// TIA Portal V17 export
// export: Created 2025-03-12T15:33:26.3402527Z, ExportSetting WithDefaults, DisplayName Totally Integrated Automation Portal, DisplayVersion V17 Update 8, DisplayName TIA Portal Openness, DisplayVersion V17 Update 8, DisplayName TIA Portal Version Control Interface, DisplayVersion V17, DisplayName SINAMICS Startdrive Advanced, DisplayVersion V17 SP2, DisplayName SINAMICS Startdrive G110M, G120, G120C, G120D, G120P, G115D, DisplayVersion V17 SP2, DisplayName SINAMICS Startdrive G130, G150, S120, S150, SINAMICS MV, S210, DisplayVersion V17 SP2, DisplayName STEP 7 Professional, DisplayVersion V17 Update 8, DisplayName SINUMERIK ONE STEP 7 Toolbox, DisplayVersion V17 Update 12, DisplayName SINUMERIK 840D sl STEP 7 Toolbox, DisplayVersion V17 Update 12, DisplayName STEP 7 Safety, DisplayVersion V17 Update 6, DisplayName WinCC Advanced, DisplayVersion V17 Update 8
FUNCTION "FC7339_ROBOT_CELL_TEST_INTERLOCK" : Void   // FC7339, LAD
{ S7_Optimized_Access := 'FALSE' }
AUTHOR : ETXETAR
VERSION : 1.0
// stored: AutoNumber false, IsIECCheckEnabled false, SetENOAutomatically false, UDAEnableTagReadback false
   VAR_TEMP
      RETVAL_1 : Int;
   END_VAR
BEGIN

REGION Network 1: ROBOT HEARTBEAT / STOP AT END OF CYCLE
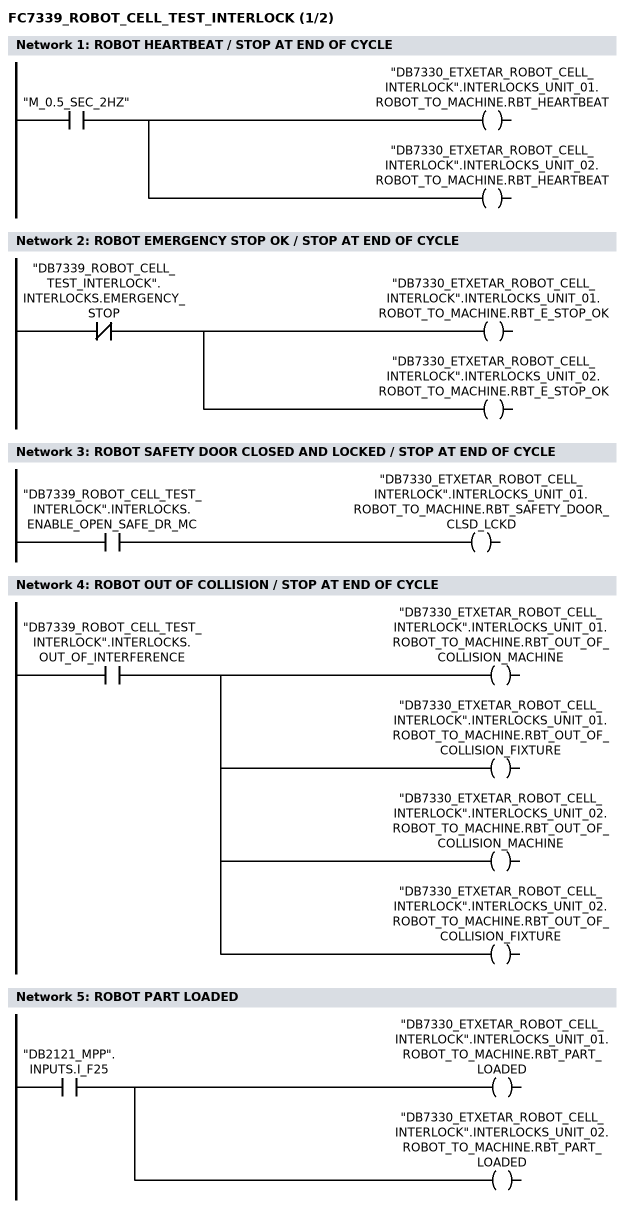
   RUNG wire#powerrail
      Contact( "M_0.5_SEC_2HZ" )
      wire#w1
      Coil( "DB7330_ETXETAR_ROBOT_CELL_INTERLOCK".INTERLOCKS_UNIT_01.ROBOT_TO_MACHINE.RBT_HEARTBEAT )
   END_RUNG
   RUNG wire#w1
      Coil( "DB7330_ETXETAR_ROBOT_CELL_INTERLOCK".INTERLOCKS_UNIT_02.ROBOT_TO_MACHINE.RBT_HEARTBEAT )
   END_RUNG
   // the same network as SCL:
   "DB7330_ETXETAR_ROBOT_CELL_INTERLOCK".INTERLOCKS_UNIT_01.ROBOT_TO_MACHINE.RBT_HEARTBEAT := "M_0.5_SEC_2HZ";
   "DB7330_ETXETAR_ROBOT_CELL_INTERLOCK".INTERLOCKS_UNIT_02.ROBOT_TO_MACHINE.RBT_HEARTBEAT := "M_0.5_SEC_2HZ";
END_REGION

REGION Network 2: ROBOT EMERGENCY STOP OK / STOP AT END OF CYCLE
   RUNG wire#powerrail
      I_Contact( "DB7339_ROBOT_CELL_TEST_INTERLOCK".INTERLOCKS.EMERGENCY_STOP )
      wire#w1
      Coil( "DB7330_ETXETAR_ROBOT_CELL_INTERLOCK".INTERLOCKS_UNIT_01.ROBOT_TO_MACHINE.RBT_E_STOP_OK )
   END_RUNG
   RUNG wire#w1
      Coil( "DB7330_ETXETAR_ROBOT_CELL_INTERLOCK".INTERLOCKS_UNIT_02.ROBOT_TO_MACHINE.RBT_E_STOP_OK )
   END_RUNG
   // the same network as SCL:
   "DB7330_ETXETAR_ROBOT_CELL_INTERLOCK".INTERLOCKS_UNIT_01.ROBOT_TO_MACHINE.RBT_E_STOP_OK := NOT "DB7339_ROBOT_CELL_TEST_INTERLOCK".INTERLOCKS.EMERGENCY_STOP;
   "DB7330_ETXETAR_ROBOT_CELL_INTERLOCK".INTERLOCKS_UNIT_02.ROBOT_TO_MACHINE.RBT_E_STOP_OK := NOT "DB7339_ROBOT_CELL_TEST_INTERLOCK".INTERLOCKS.EMERGENCY_STOP;
END_REGION

REGION Network 3: ROBOT SAFETY DOOR CLOSED AND LOCKED / STOP AT END OF CYCLE
   RUNG wire#powerrail
      Contact( "DB7339_ROBOT_CELL_TEST_INTERLOCK".INTERLOCKS.ENABLE_OPEN_SAFE_DR_MC )
      Coil( "DB7330_ETXETAR_ROBOT_CELL_INTERLOCK".INTERLOCKS_UNIT_01.ROBOT_TO_MACHINE.RBT_SAFETY_DOOR_CLSD_LCKD )
   END_RUNG
   // the same network as SCL:
   "DB7330_ETXETAR_ROBOT_CELL_INTERLOCK".INTERLOCKS_UNIT_01.ROBOT_TO_MACHINE.RBT_SAFETY_DOOR_CLSD_LCKD := "DB7339_ROBOT_CELL_TEST_INTERLOCK".INTERLOCKS.ENABLE_OPEN_SAFE_DR_MC;
END_REGION

REGION Network 4: ROBOT OUT OF COLLISION / STOP AT END OF CYCLE
   RUNG wire#powerrail
      Contact( "DB7339_ROBOT_CELL_TEST_INTERLOCK".INTERLOCKS.OUT_OF_INTERFERENCE )
      wire#w1
      Coil( "DB7330_ETXETAR_ROBOT_CELL_INTERLOCK".INTERLOCKS_UNIT_01.ROBOT_TO_MACHINE.RBT_OUT_OF_COLLISION_MACHINE )
   END_RUNG
   RUNG wire#w1
      Coil( "DB7330_ETXETAR_ROBOT_CELL_INTERLOCK".INTERLOCKS_UNIT_01.ROBOT_TO_MACHINE.RBT_OUT_OF_COLLISION_FIXTURE )
   END_RUNG
   RUNG wire#w1
      Coil( "DB7330_ETXETAR_ROBOT_CELL_INTERLOCK".INTERLOCKS_UNIT_02.ROBOT_TO_MACHINE.RBT_OUT_OF_COLLISION_MACHINE )
   END_RUNG
   RUNG wire#w1
      Coil( "DB7330_ETXETAR_ROBOT_CELL_INTERLOCK".INTERLOCKS_UNIT_02.ROBOT_TO_MACHINE.RBT_OUT_OF_COLLISION_FIXTURE )
   END_RUNG
   // the same network as SCL:
   "DB7330_ETXETAR_ROBOT_CELL_INTERLOCK".INTERLOCKS_UNIT_01.ROBOT_TO_MACHINE.RBT_OUT_OF_COLLISION_MACHINE := "DB7339_ROBOT_CELL_TEST_INTERLOCK".INTERLOCKS.OUT_OF_INTERFERENCE;
   "DB7330_ETXETAR_ROBOT_CELL_INTERLOCK".INTERLOCKS_UNIT_01.ROBOT_TO_MACHINE.RBT_OUT_OF_COLLISION_FIXTURE := "DB7339_ROBOT_CELL_TEST_INTERLOCK".INTERLOCKS.OUT_OF_INTERFERENCE;
   "DB7330_ETXETAR_ROBOT_CELL_INTERLOCK".INTERLOCKS_UNIT_02.ROBOT_TO_MACHINE.RBT_OUT_OF_COLLISION_MACHINE := "DB7339_ROBOT_CELL_TEST_INTERLOCK".INTERLOCKS.OUT_OF_INTERFERENCE;
   "DB7330_ETXETAR_ROBOT_CELL_INTERLOCK".INTERLOCKS_UNIT_02.ROBOT_TO_MACHINE.RBT_OUT_OF_COLLISION_FIXTURE := "DB7339_ROBOT_CELL_TEST_INTERLOCK".INTERLOCKS.OUT_OF_INTERFERENCE;
END_REGION

REGION Network 5: ROBOT PART LOADED
   RUNG wire#powerrail
      Contact( "DB2121_MPP".INPUTS.I_F25 )
      wire#w1
      Coil( "DB7330_ETXETAR_ROBOT_CELL_INTERLOCK".INTERLOCKS_UNIT_01.ROBOT_TO_MACHINE.RBT_PART_LOADED )
   END_RUNG
   RUNG wire#w1
      Coil( "DB7330_ETXETAR_ROBOT_CELL_INTERLOCK".INTERLOCKS_UNIT_02.ROBOT_TO_MACHINE.RBT_PART_LOADED )
   END_RUNG
   // the same network as SCL:
   "DB7330_ETXETAR_ROBOT_CELL_INTERLOCK".INTERLOCKS_UNIT_01.ROBOT_TO_MACHINE.RBT_PART_LOADED := "DB2121_MPP".INPUTS.I_F25;
   "DB7330_ETXETAR_ROBOT_CELL_INTERLOCK".INTERLOCKS_UNIT_02.ROBOT_TO_MACHINE.RBT_PART_LOADED := "DB2121_MPP".INPUTS.I_F25;
END_REGION

REGION Network 6: ROBOT PART UNLOADED
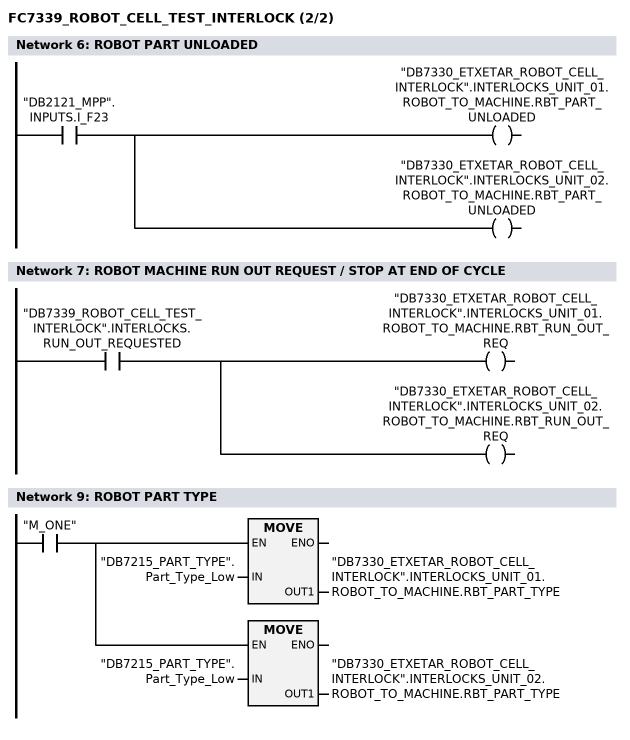
   RUNG wire#powerrail
      Contact( "DB2121_MPP".INPUTS.I_F23 )
      wire#w1
      Coil( "DB7330_ETXETAR_ROBOT_CELL_INTERLOCK".INTERLOCKS_UNIT_01.ROBOT_TO_MACHINE.RBT_PART_UNLOADED )
   END_RUNG
   RUNG wire#w1
      Coil( "DB7330_ETXETAR_ROBOT_CELL_INTERLOCK".INTERLOCKS_UNIT_02.ROBOT_TO_MACHINE.RBT_PART_UNLOADED )
   END_RUNG
   // the same network as SCL:
   "DB7330_ETXETAR_ROBOT_CELL_INTERLOCK".INTERLOCKS_UNIT_01.ROBOT_TO_MACHINE.RBT_PART_UNLOADED := "DB2121_MPP".INPUTS.I_F23;
   "DB7330_ETXETAR_ROBOT_CELL_INTERLOCK".INTERLOCKS_UNIT_02.ROBOT_TO_MACHINE.RBT_PART_UNLOADED := "DB2121_MPP".INPUTS.I_F23;
END_REGION

REGION Network 7: ROBOT MACHINE RUN OUT REQUEST / STOP AT END OF CYCLE
   RUNG wire#powerrail
      Contact( "DB7339_ROBOT_CELL_TEST_INTERLOCK".INTERLOCKS.RUN_OUT_REQUESTED )
      wire#w1
      Coil( "DB7330_ETXETAR_ROBOT_CELL_INTERLOCK".INTERLOCKS_UNIT_01.ROBOT_TO_MACHINE.RBT_RUN_OUT_REQ )
   END_RUNG
   RUNG wire#w1
      Coil( "DB7330_ETXETAR_ROBOT_CELL_INTERLOCK".INTERLOCKS_UNIT_02.ROBOT_TO_MACHINE.RBT_RUN_OUT_REQ )
   END_RUNG
   // the same network as SCL:
   "DB7330_ETXETAR_ROBOT_CELL_INTERLOCK".INTERLOCKS_UNIT_01.ROBOT_TO_MACHINE.RBT_RUN_OUT_REQ := "DB7339_ROBOT_CELL_TEST_INTERLOCK".INTERLOCKS.RUN_OUT_REQUESTED;
   "DB7330_ETXETAR_ROBOT_CELL_INTERLOCK".INTERLOCKS_UNIT_02.ROBOT_TO_MACHINE.RBT_RUN_OUT_REQ := "DB7339_ROBOT_CELL_TEST_INTERLOCK".INTERLOCKS.RUN_OUT_REQUESTED;
END_REGION

REGION Network 8: ROBOT PART TYPE CHANGE REQUEST / STOP AT END OF CYCLE
END_REGION

REGION Network 9: ROBOT PART TYPE
   RUNG wire#powerrail
      Contact( "M_ONE" )
      wire#w1
      Move(in := "DB7215_PART_TYPE".Part_Type_Low, out1 => "DB7330_ETXETAR_ROBOT_CELL_INTERLOCK".INTERLOCKS_UNIT_01.ROBOT_TO_MACHINE.RBT_PART_TYPE)
   END_RUNG
   RUNG wire#w1
      Move(in := "DB7215_PART_TYPE".Part_Type_Low, out1 => "DB7330_ETXETAR_ROBOT_CELL_INTERLOCK".INTERLOCKS_UNIT_02.ROBOT_TO_MACHINE.RBT_PART_TYPE)
   END_RUNG
   // the same network as SCL:
   IF "M_ONE" THEN
       "DB7330_ETXETAR_ROBOT_CELL_INTERLOCK".INTERLOCKS_UNIT_01.ROBOT_TO_MACHINE.RBT_PART_TYPE := "DB7215_PART_TYPE".Part_Type_Low;
       "DB7330_ETXETAR_ROBOT_CELL_INTERLOCK".INTERLOCKS_UNIT_02.ROBOT_TO_MACHINE.RBT_PART_TYPE := "DB7215_PART_TYPE".Part_Type_Low;
   END_IF;
END_REGION
END_FUNCTION
